TYPE ZDataMachine :
STRUCT
{region "Scribly"}
{IF NOT (defined (Scribly_disabled))}
  Scribly : ScriblyDataMachine;
  {attribute 'ZId' := '61e5b130-0fef-4d8b-85dd-afb1efcde47c'}
{END_IF}
{endregion}
{attribute '__ZwPlcApplicationDataMachineDeclaration__'} // Do not remove this attribute! It is used for code generation.
END_STRUCT
END_TYPE

(* stored: Version 1.1.0.1
   DUT ZDataMachine: Id {48717368-9a5e-4668-a675-3da0af6e27e0} *)
